FUNCTION_BLOCK VBT IMPLEMENTS MachineModule
VAR
	bEnable			: BOOL;
	bDisable        : BOOL;
	bError          : BOOL;
	bOverride       : BOOL;
	bSimulation     : BOOL;
	bStart          : BOOL;
	bStop           : BOOL;
END_VAR

// This is the core module needed that we are creating for our STS and contains everything related to the STS

// To be added
(*
FEEDER

SAT

VBT

EJECT

GATE

SBT

*)

METHOD Disable : BOOL
VAR_INPUT
END_VAR
bEnable:=FALSE;
END_METHOD

METHOD Enable : BOOL
VAR_INPUT
END_VAR
bEnable:=TRUE;
bDisable:=False;
END_METHOD

METHOD Error : BOOL
VAR_INPUT
END_VAR
bEnable:=FALSE;
END_METHOD

METHOD Override : BOOL
VAR_INPUT
END_VAR
END_METHOD

METHOD Start : BOOL
VAR_INPUT
END_VAR
END_METHOD

METHOD PUBLIC StateMachine
VAR_INPUT
END_VAR
END_METHOD

METHOD Stop : BOOL
VAR_INPUT
END_VAR
END_METHOD

END_FUNCTION_BLOCK

(* stored: Version 1.1.0.1, ProductVersion 3.1.4024.12
   POU VBT: Id {cec5e054-0329-4fa9-83b2-adb3800b30c6}, SpecialFunc None
   Method Disable: Id {945decf1-cc3b-4249-bcf7-a5ed9082fc2f}
   Method Enable: Id {8b4709de-56a3-4871-8de2-ce3de4c3d3f3}
   Method Error: Id {b50cb842-6df4-4043-b5c5-ed9e5d560ad8}
   Method Override: Id {4de31e82-6ee8-433f-8e5d-89f9b09e6bc8}
   Method Start: Id {df34af96-b1fb-41af-b3f5-4280fcd2af5f}
   Method StateMachine: Id {dc2d00cb-2e39-4ebc-915b-dbf5c98e2b23}
   Method Stop: Id {76b10ce9-f27e-4523-814b-cf31943a6760} *)
